(* Logix 5000 project; controller Tekno_ASRS vendor 1 type 14 code 147 rev 20.11; software revision 20.01; part 2 of 4 *)
(* tags used below, declared in another part *)
   AAxis : AXIS_CIP_DRIVE;
   AAxisMAM : MOTION_INSTRUCTION;
   AAxisMove : BOOL;
   AAxisOn : MOTION_INSTRUCTION;
   AAXisReset : MOTION_INSTRUCTION;
   AftAreaScanner : DCI_STOP;
   AftAreaZn2 : ALIAS FOR ShuttleIO:10:O.2;
   AftEndZn : BOOL;
   AftEndZnLimit : DINT;
   AftEndZone : BOOL;
   AgridLoc : DINT;
   AGVatDP : ALIAS FOR StationaryIO:1:I.3;
   AGVatPU : ALIAS FOR StationaryIO:1:I.2;
   AGVok2LvDP : ALIAS FOR StationaryIO:8:O.0;
   AGVok2LvPU : ALIAS FOR StationaryIO:8:O.1;
   AreaWarn : ALIAS FOR ShuttleIO:5:O.2;
   ASRSEnable : BOOL;
   ASRSMCR : BOOL;
   ASRSStatus : ASRS_Status;
   AutoConfig : Configuration;
   AxisStateReady : BOOL;
   BackGateInstalled : ALIAS FOR ShuttleIO:9:I.Pt01Data;
   BAxis : AXIS_CIP_DRIVE;
   BAxisMAM : MOTION_INSTRUCTION;
   BAxisMove : BOOL;
   BAXisReset : MOTION_INSTRUCTION;
   BgridLoc : DINT;
   BrakeTmr : TIMER;
   CCoordSetup : BOOL;
   CfgEnd : BayPos;
   CfgStrt : BayPos;
   CGridLoc : DINT;
   Configuration : Configuration;
   CurrentAPos : DINT;
   CurrentBPos : DINT;
   CurrentCPos : DINT;
   CurrentTask : Task;
   DemoDP : Task[3];
   DemoOns : BOOL;
   DemoPU : Task[3];
   DPCntr : DINT;
   DPReg : BOOL;
   DriveEnabled : BOOL;
   DrivesOn : BOOL;
   EStop_SafetyGate : DCI_STOP;
   FootSwitch : ALIAS FOR ShuttleIO:9:I.Pt04Data;
   ForeAreaScanner : DCI_STOP;
   ForeAreaZn2 : ALIAS FOR ShuttleIO:10:O.0;
   FrntAreaWarn : ALIAS FOR ShuttleIO:9:I.Pt00Data;
   FwdEndZn : BOOL;
   FwdEndZone : BOOL;
   GZSet : BOOL;
   GZSetEnable : BOOL;
   HighSpeedFwd : BOOL;
   HighSpeedRev : BOOL;
   HMI_Commands : HMI_Commands;
   HMIData : HMI_Data;
   HMIMsgCtrl : MESSAGE;
   HMITmr : TIMER;
   HomeSpatula : BOOL;
   Horn : ALIAS FOR ShuttleIO:5:O.1;
   JogAAxisEn : BOOL;
   JogActive : BOOL;
   JogARev : BOOL;
   JogBAxisEn : BOOL;
   JogReleaseSBrk : BOOL;
   LastAAxFlt : DINT;
   LastBAxFlt : DINT;
   LastMessageReceiveSequence : DINT;
   LiftStrainFault : BOOL;
   LiftStrainOK : BOOL;
   LoadaTask : BOOL;
   LoadTask : Task;
   LockRelease : ALIAS FOR StationaryIO:7:I.Pt04Data;
   ManConfig : Configuration;
   ManGateClosed : ALIAS FOR ShuttleIO:9:I.Pt02Data;
   ManMode : BOOL;
   ManOnBoard : ALIAS FOR ShuttleIO:5:O.5;
   MasterReset : BOOL;
   MatrixSetup : BOOL;
   MaxA : DINT;
   MaxB : DINT;
   MaxC : DINT;
   MoveComplete : BOOL;
   MoveInProcess : BOOL;
   MoveRequested : BOOL;
   MoveSafetyEnable : BOOL;
   NewAPos : DINT;
   NewBPos : DINT;
   NewCmnd : DINT;
   NewCPos : DINT;
   Override : BOOL;
   PalmButtonLeft : ALIAS FOR ShuttleIO:9:I.Pt07Data;
   PalmButtonRight : ALIAS FOR ShuttleIO:9:I.Pt06Data;
   PalmButtons : DCI_STOP;
   PorDInProc : BOOL;
   PorDStop : BOOL;
   PositionFlt : BOOL;
   PUCntr : DINT;
   Pulse : TIMER;
   PulseBit : BOOL;
   PUReg : BOOL;
   RearAreaWarn : ALIAS FOR ShuttleIO:9:I.Pt05Data;
   ReceiveMessage : Messaging;
   ReleaseSpatBrk : BOOL;
   ResetTmr : TIMER;
   RowObstruction : BOOL;
   RPE_400140 : ALIAS FOR StationaryIO:2:I.0;
   RPE_400150 : ALIAS FOR StationaryIO:2:I.1;
   RPE_400160 : ALIAS FOR StationaryIO:2:I.2;
   RPE_400170 : ALIAS FOR StationaryIO:2:I.3;
   RPE_400180 : ALIAS FOR StationaryIO:2:I.4;
   RPE_400190 : ALIAS FOR StationaryIO:2:I.5;
   RPE_400200 : ALIAS FOR StationaryIO:2:I.6;
   RPE_400210 : ALIAS FOR StationaryIO:2:I.7;
   RPE_400280 : ALIAS FOR StationaryIO:3:I.0;
   RPE_400290 : ALIAS FOR StationaryIO:3:I.1;
   RPE_400300 : ALIAS FOR StationaryIO:3:I.2;
   RPE_400310 : ALIAS FOR StationaryIO:3:I.3;
   RPE_400320 : ALIAS FOR StationaryIO:3:I.4;
   RPE_400330 : ALIAS FOR StationaryIO:3:I.5;
   RPE_400340 : ALIAS FOR StationaryIO:3:I.6;
   RPE_400350 : ALIAS FOR StationaryIO:3:I.7;
   RPE_400390 : ALIAS FOR StationaryIO:4:I.0;
   RPE_400400 : ALIAS FOR StationaryIO:4:I.1;
   RPE_400410 : ALIAS FOR StationaryIO:4:I.2;
   SafetyReset : ALIAS FOR StationaryIO:7:I.Pt03Data;
   ShuttleFault : ALIAS FOR ShuttleIO:5:O.3;
   SpatulaBrake : ALIAS FOR ShuttleIO:5:O.6;
   SpatulaHome : ALIAS FOR ShuttleIO:2:I.4;
   Start : ALIAS FOR StationaryIO:7:I.Pt02Data;
   StationaryFlt : BOOL;
   StationaryHrn : BOOL;
   StationaryMnOn : BOOL;
   StationaryRn : BOOL;
   StationaryWrn : BOOL;
   Stop : ALIAS FOR StationaryIO:7:I.Pt05Data;
   StrainFltTtl : DINT;
   SUIndPos : BOOL;
   SystemRunning : ALIAS FOR ShuttleIO:5:O.0;
   TaskFIFO : CONTROL;
   TaskFile : Task[100];
   TaskInProcess : BOOL;
   TestRun : Task[20];
   TestStop : BOOL;
   UnBindInProc : BOOL;
   XAxisBrk : ALIAS FOR ShuttleIO:5:O.4;
   XAxisEOTFlt : BOOL;
   XAxisMtrSideEOT : ALIAS FOR ShuttleIO:2:I.6;
   XAxisPnlSideEOT : ALIAS FOR ShuttleIO:2:I.7;
   XBrakeTmr : TIMER;
   XLtCTTmr : TIMER;
   XLtTTmr : TIMER;
   XPosHoldTmr : TIMER;
   XRtCTTmr : TIMER;
   XRtTTmr : TIMER;
   XStCalMode : ALIAS FOR StationaryIO:5:O.Data[0].0;
   XStrain : Strain;
   XStRunMode : ALIAS FOR StationaryIO:5:O.Data[0].1;
   XTensionOK : BOOL;
   ZAftLeftOK : BOOL;
   ZAftLtCTTmr : TIMER;
   ZAftLtTTmr : TIMER;
   ZAftRightOK : BOOL;
   ZAftRtCTTmr : TIMER;
   ZAftRtTTmr : TIMER;
   ZAftStCalMode : ALIAS FOR ShuttleIO:4:O.Data[0].0;
   ZAftStrain : Strain;
   ZAftStRunMode : ALIAS FOR ShuttleIO:4:O.Data[0].1;
   ZAxisBrk : ALIAS FOR ShuttleIO:5:O.7;
   ZAxisDnEOT : ALIAS FOR ShuttleIO:1:I.1;
   ZAxisEOTFlt : BOOL;
   ZAxisSafetyDisengage : BOOL;
   ZAxisUpEOT : ALIAS FOR ShuttleIO:1:I.0;
   ZForeLeftOK : BOOL;
   ZForeRightOK : BOOL;
   ZForeStCalMode : ALIAS FOR ShuttleIO:3:O.Data[0].0;
   ZForeStrain : Strain;
   ZForeStRunMode : ALIAS FOR ShuttleIO:3:O.Data[0].1;
   ZForLtCTTmr : TIMER;
   ZForLtTTmr : TIMER;
   ZForRtCTTmr : TIMER;
   ZForRtTTmr : TIMER;
   ZLAftLft : ALIAS FOR ShuttleIO:2:I.0;
   ZLAftRgt : ALIAS FOR ShuttleIO:2:I.1;
   ZLAutoDly : DINT;
   ZLBindTmr : TIMER;
   ZLFault : BOOL;
   ZLForeLft : ALIAS FOR ShuttleIO:2:I.3;
   ZLForeRgt : ALIAS FOR ShuttleIO:2:I.2;
   ZLManDly : DINT;
   ZLockDelay : TIMER;
   ZLsDisengaged : BOOL;
   ZLsProxOK : BOOL;
   ZPosHoldTmr : TIMER;

PROGRAM MainProgram   (* main routine MainRoutine *)
VAR
   AAxisOff : MOTION_INSTRUCTION := (FLAGS := 536870912, DN := 1, STATUS := 2, STATE := 1);
   AAxisStateMask : DINT;
   AutoMode : BOOL;
   BAxisOff : MOTION_INSTRUCTION := (FLAGS := 536870912, DN := 1, STATUS := 2, STATE := 1);
   BAxisStateMask : DINT;
   msgtest : BOOL;
   msgtest2 : BOOL;
END_VAR

ROUTINE HMI   (* ladder *)
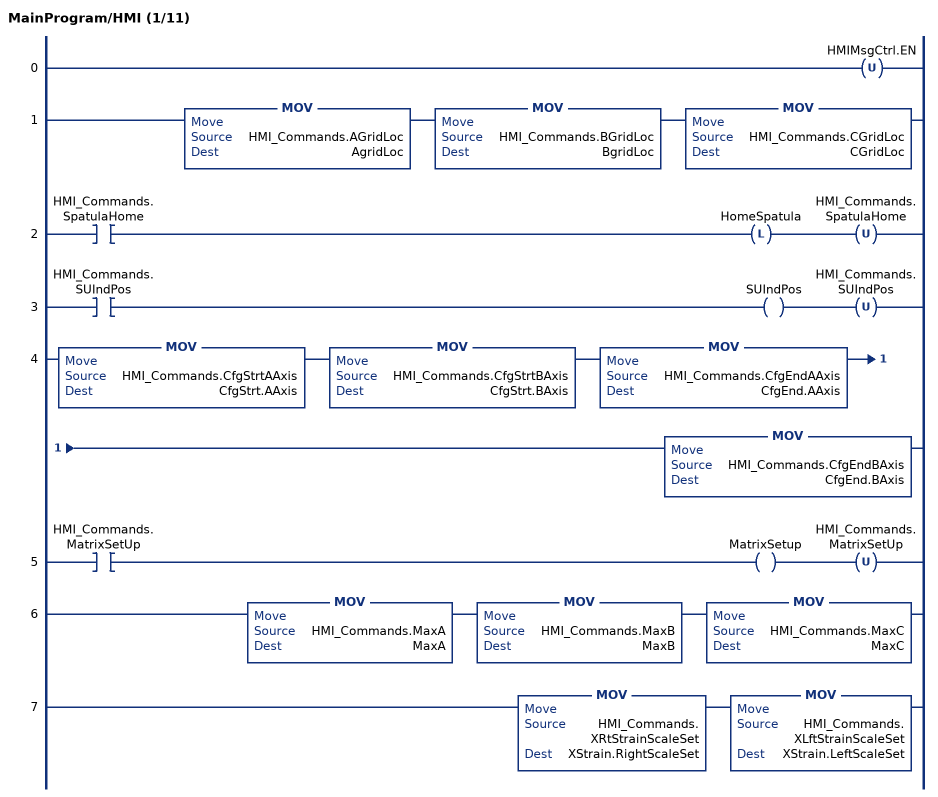
   0: OTU(HMIMsgCtrl.EN);
   1: MOV(HMI_Commands.AGridLoc,AgridLoc)MOV(HMI_Commands.BGridLoc,BgridLoc)MOV(HMI_Commands.CGridLoc,CGridLoc);
   2: XIC(HMI_Commands.SpatulaHome)OTL(HomeSpatula)OTU(HMI_Commands.SpatulaHome);
   3: XIC(HMI_Commands.SUIndPos)OTE(SUIndPos)OTU(HMI_Commands.SUIndPos);
   4: MOV(HMI_Commands.CfgStrtAAxis,CfgStrt.AAxis)MOV(HMI_Commands.CfgStrtBAxis,CfgStrt.BAxis)MOV(HMI_Commands.CfgEndAAxis,CfgEnd.AAxis)MOV(HMI_Commands.CfgEndBAxis,CfgEnd.BAxis);
   5: XIC(HMI_Commands.MatrixSetUp)OTE(MatrixSetup)OTU(HMI_Commands.MatrixSetUp);
   6: MOV(HMI_Commands.MaxA,MaxA)MOV(HMI_Commands.MaxB,MaxB)MOV(HMI_Commands.MaxC,MaxC);
   7: MOV(HMI_Commands.XRtStrainScaleSet,XStrain.RightScaleSet)MOV(HMI_Commands.XLftStrainScaleSet,XStrain.LeftScaleSet);
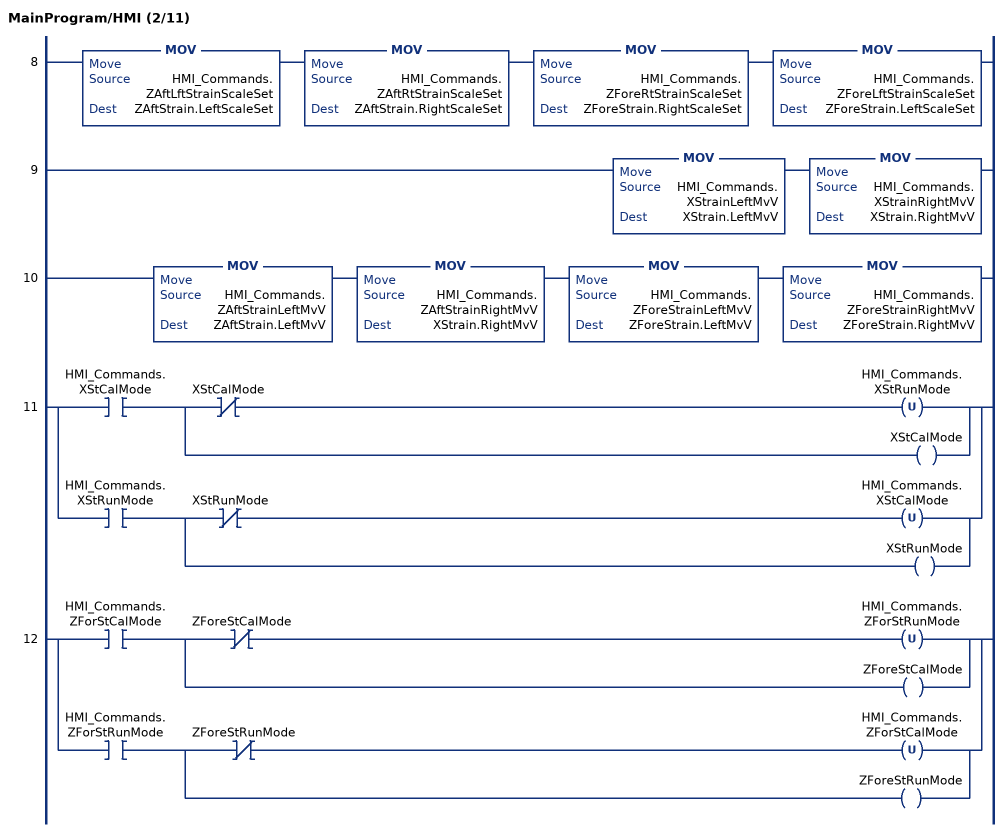
   8: MOV(HMI_Commands.ZAftLftStrainScaleSet,ZAftStrain.LeftScaleSet)MOV(HMI_Commands.ZAftRtStrainScaleSet,ZAftStrain.RightScaleSet)MOV(HMI_Commands.ZForeRtStrainScaleSet,ZForeStrain.RightScaleSet)MOV(HMI_Commands.ZForeLftStrainScaleSet,ZForeStrain.LeftScaleSet);
   9: MOV(HMI_Commands.XStrainLeftMvV,XStrain.LeftMvV)MOV(HMI_Commands.XStrainRightMvV,XStrain.RightMvV);
   10: MOV(HMI_Commands.ZAftStrainLeftMvV,ZAftStrain.LeftMvV)MOV(HMI_Commands.ZAftStrainRightMvV,XStrain.RightMvV)MOV(HMI_Commands.ZForeStrainLeftMvV,ZForeStrain.LeftMvV)MOV(HMI_Commands.ZForeStrainRightMvV,ZForeStrain.RightMvV);
   11: [XIC(HMI_Commands.XStCalMode) [XIO(XStCalMode) OTU(HMI_Commands.XStRunMode) ,OTE(XStCalMode) ] ,XIC(HMI_Commands.XStRunMode) [XIO(XStRunMode) OTU(HMI_Commands.XStCalMode) ,OTE(XStRunMode) ] ];
   12: [XIC(HMI_Commands.ZForStCalMode) [XIO(ZForeStCalMode) OTU(HMI_Commands.ZForStRunMode) ,OTE(ZForeStCalMode) ] ,XIC(HMI_Commands.ZForStRunMode) [XIO(ZForeStRunMode) OTU(HMI_Commands.ZForStCalMode) ,OTE(ZForeStRunMode) ] ];
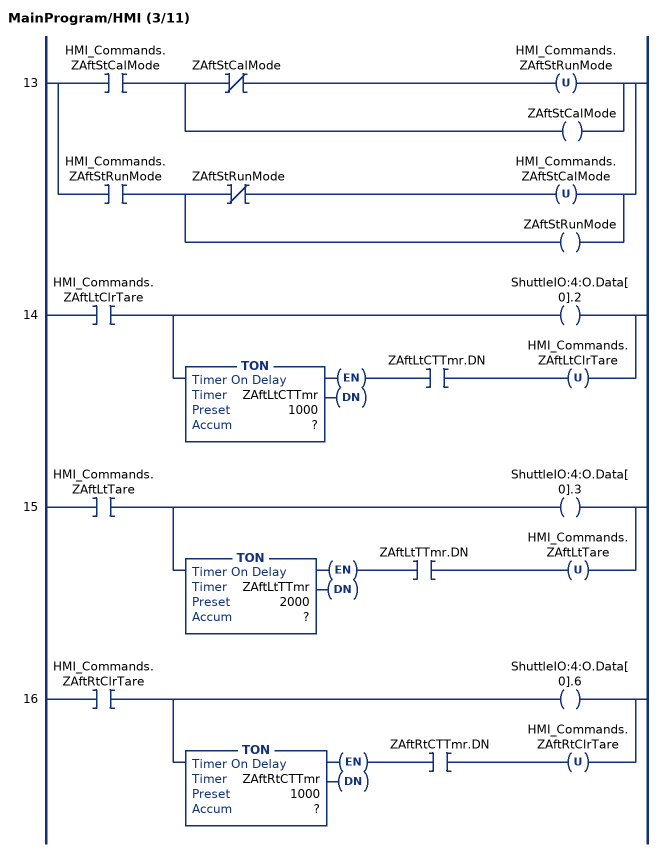
   13: [XIC(HMI_Commands.ZAftStCalMode) [XIO(ZAftStCalMode) OTU(HMI_Commands.ZAftStRunMode) ,OTE(ZAftStCalMode) ] ,XIC(HMI_Commands.ZAftStRunMode) [XIO(ZAftStRunMode) OTU(HMI_Commands.ZAftStCalMode) ,OTE(ZAftStRunMode) ] ];
   14: XIC(HMI_Commands.ZAftLtClrTare)[OTE(ShuttleIO:4:O.Data[0].2) ,TON(ZAftLtCTTmr,?,?) XIC(ZAftLtCTTmr.DN) OTU(HMI_Commands.ZAftLtClrTare) ];
   15: XIC(HMI_Commands.ZAftLtTare)[OTE(ShuttleIO:4:O.Data[0].3) ,TON(ZAftLtTTmr,?,?) XIC(ZAftLtTTmr.DN) OTU(HMI_Commands.ZAftLtTare) ];
   16: XIC(HMI_Commands.ZAftRtClrTare)[OTE(ShuttleIO:4:O.Data[0].6) ,TON(ZAftRtCTTmr,?,?) XIC(ZAftRtCTTmr.DN) OTU(HMI_Commands.ZAftRtClrTare) ];
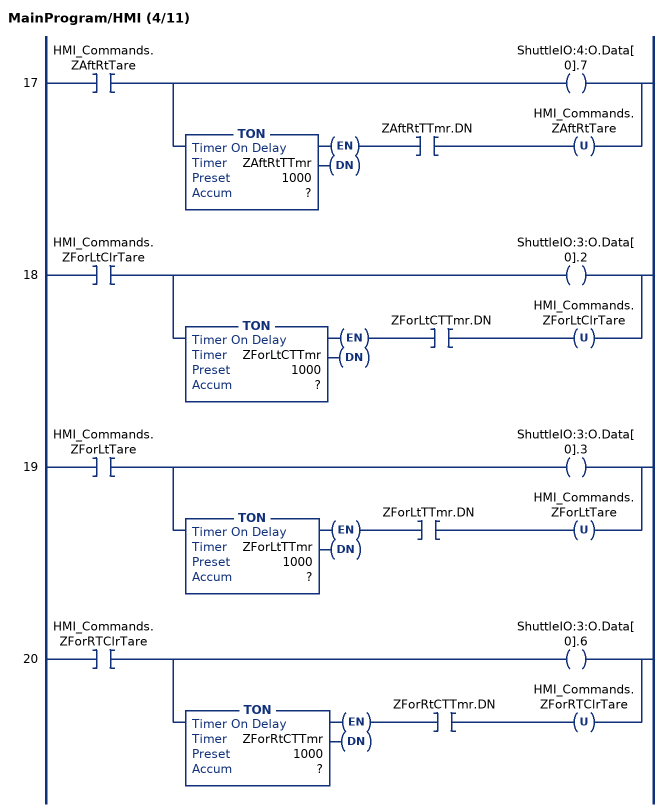
   17: XIC(HMI_Commands.ZAftRtTare)[OTE(ShuttleIO:4:O.Data[0].7) ,TON(ZAftRtTTmr,?,?) XIC(ZAftRtTTmr.DN) OTU(HMI_Commands.ZAftRtTare) ];
   18: XIC(HMI_Commands.ZForLtClrTare)[OTE(ShuttleIO:3:O.Data[0].2) ,TON(ZForLtCTTmr,?,?) XIC(ZForLtCTTmr.DN) OTU(HMI_Commands.ZForLtClrTare) ];
   19: XIC(HMI_Commands.ZForLtTare)[OTE(ShuttleIO:3:O.Data[0].3) ,TON(ZForLtTTmr,?,?) XIC(ZForLtTTmr.DN) OTU(HMI_Commands.ZForLtTare) ];
   20: XIC(HMI_Commands.ZForRTClrTare)[OTE(ShuttleIO:3:O.Data[0].6) ,TON(ZForRtCTTmr,?,?) XIC(ZForRtCTTmr.DN) OTU(HMI_Commands.ZForRTClrTare) ];
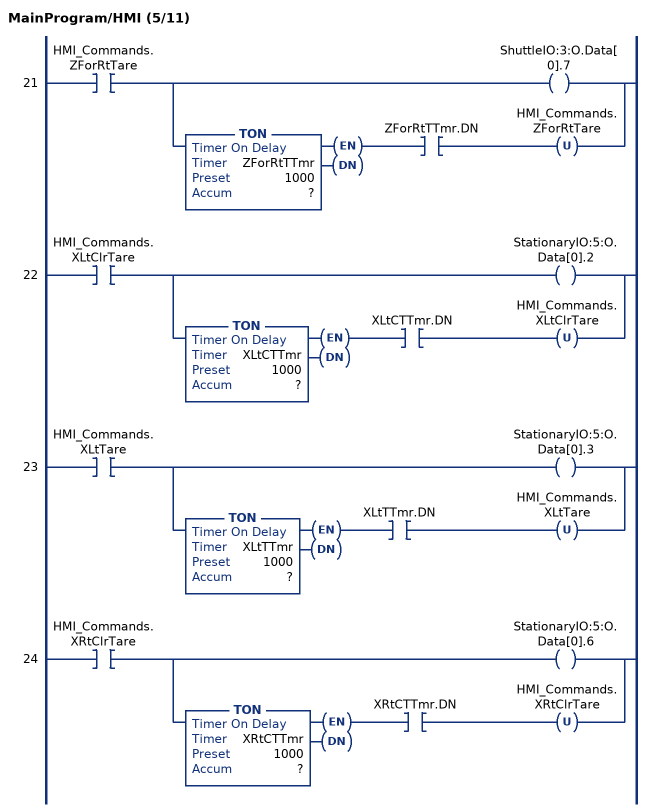
   21: XIC(HMI_Commands.ZForRtTare)[OTE(ShuttleIO:3:O.Data[0].7) ,TON(ZForRtTTmr,?,?) XIC(ZForRtTTmr.DN) OTU(HMI_Commands.ZForRtTare) ];
   22: XIC(HMI_Commands.XLtClrTare)[OTE(StationaryIO:5:O.Data[0].2) ,TON(XLtCTTmr,?,?) XIC(XLtCTTmr.DN) OTU(HMI_Commands.XLtClrTare) ];
   23: XIC(HMI_Commands.XLtTare)[OTE(StationaryIO:5:O.Data[0].3) ,TON(XLtTTmr,?,?) XIC(XLtTTmr.DN) OTU(HMI_Commands.XLtTare) ];
   24: XIC(HMI_Commands.XRtClrTare)[OTE(StationaryIO:5:O.Data[0].6) ,TON(XRtCTTmr,?,?) XIC(XRtCTTmr.DN) OTU(HMI_Commands.XRtClrTare) ];
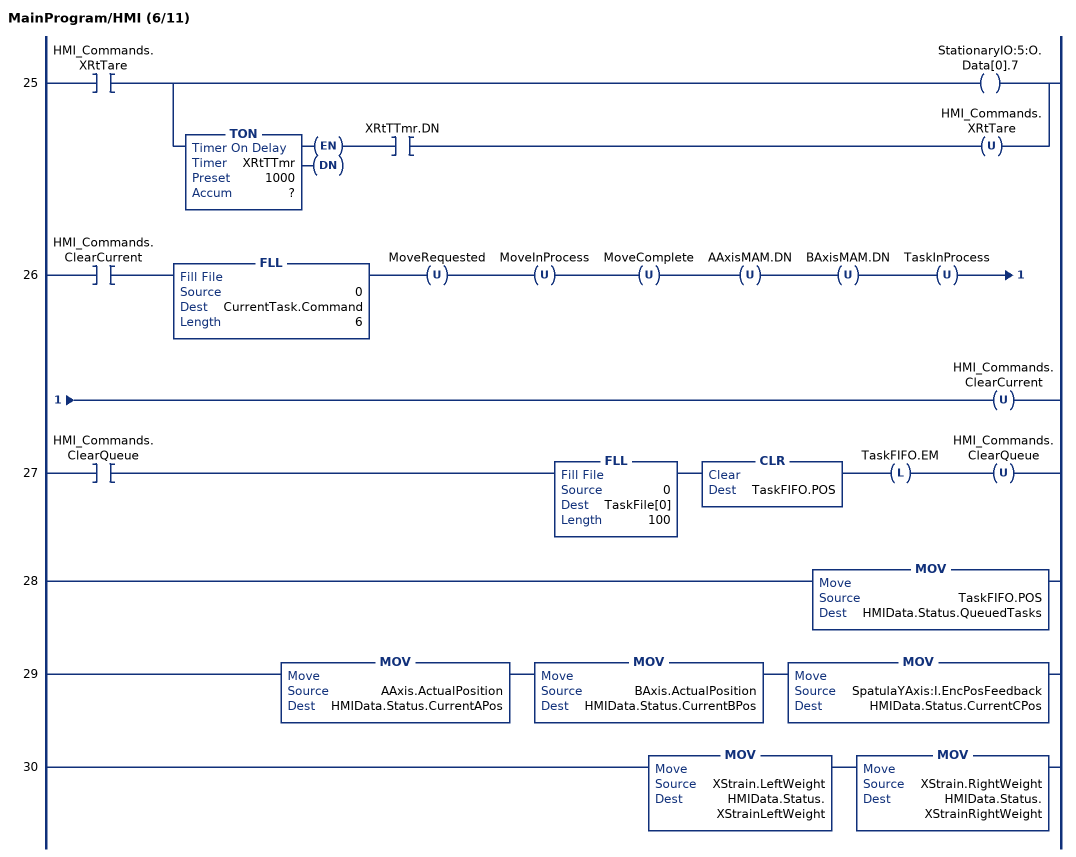
   25: XIC(HMI_Commands.XRtTare)[OTE(StationaryIO:5:O.Data[0].7) ,TON(XRtTTmr,?,?) XIC(XRtTTmr.DN) OTU(HMI_Commands.XRtTare) ];
   26: XIC(HMI_Commands.ClearCurrent)FLL(0,CurrentTask.Command,6)OTU(MoveRequested)OTU(MoveInProcess)OTU(MoveComplete)OTU(AAxisMAM.DN)OTU(BAxisMAM.DN)OTU(TaskInProcess)OTU(HMI_Commands.ClearCurrent);
   27: XIC(HMI_Commands.ClearQueue)FLL(0,TaskFile[0],100)CLR(TaskFIFO.POS)OTL(TaskFIFO.EM)OTU(HMI_Commands.ClearQueue);
   28: MOV(TaskFIFO.POS,HMIData.Status.QueuedTasks);
   29: MOV(AAxis.ActualPosition,HMIData.Status.CurrentAPos)MOV(BAxis.ActualPosition,HMIData.Status.CurrentBPos)MOV(SpatulaYAxis:I.EncPosFeedback,HMIData.Status.CurrentCPos);
   30: MOV(XStrain.LeftWeight,HMIData.Status.XStrainLeftWeight)MOV(XStrain.RightWeight,HMIData.Status.XStrainRightWeight);
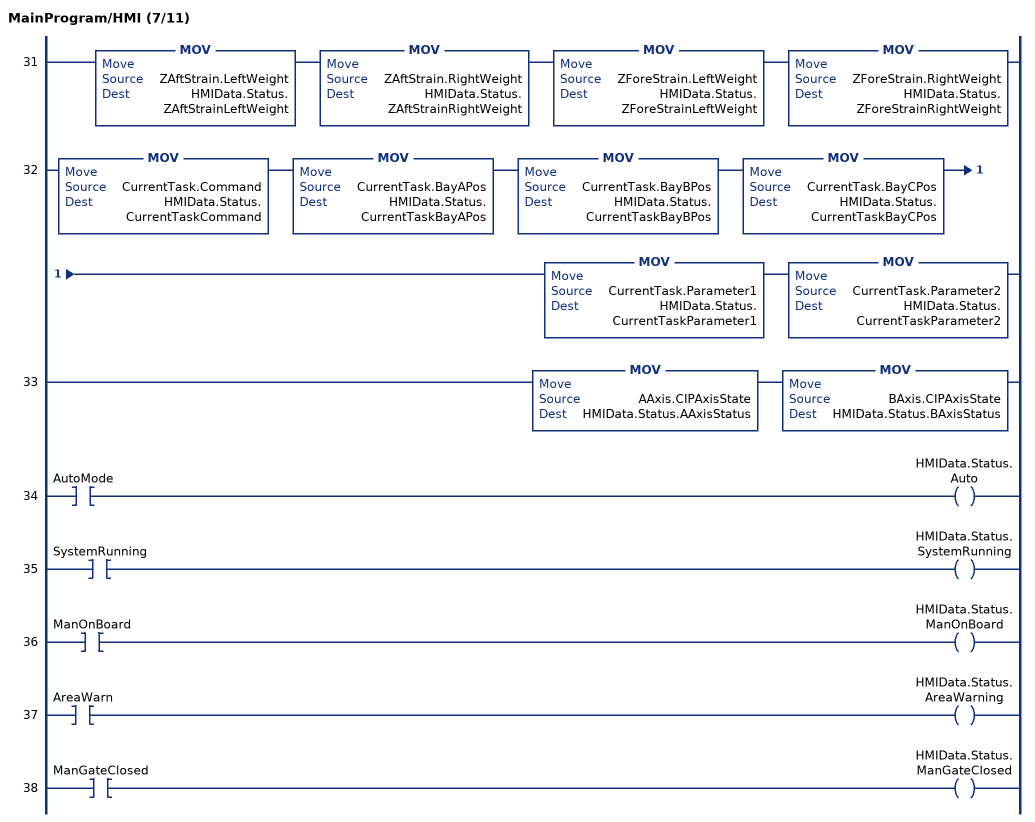
   31: MOV(ZAftStrain.LeftWeight,HMIData.Status.ZAftStrainLeftWeight)MOV(ZAftStrain.RightWeight,HMIData.Status.ZAftStrainRightWeight)MOV(ZForeStrain.LeftWeight,HMIData.Status.ZForeStrainLeftWeight)MOV(ZForeStrain.RightWeight,HMIData.Status.ZForeStrainRightWeight);
   32: MOV(CurrentTask.Command,HMIData.Status.CurrentTaskCommand)MOV(CurrentTask.BayAPos,HMIData.Status.CurrentTaskBayAPos)MOV(CurrentTask.BayBPos,HMIData.Status.CurrentTaskBayBPos)MOV(CurrentTask.BayCPos,HMIData.Status.CurrentTaskBayCPos)MOV(CurrentTask.Parameter1,HMIData.Status.CurrentTaskParameter1)MOV(CurrentTask.Parameter2,HMIData.Status.CurrentTaskParameter2);
   33: MOV(AAxis.CIPAxisState,HMIData.Status.AAxisStatus)MOV(BAxis.CIPAxisState,HMIData.Status.BAxisStatus);
   34: XIC(AutoMode)OTE(HMIData.Status.Auto);
   35: XIC(SystemRunning)OTE(HMIData.Status.SystemRunning);
   36: XIC(ManOnBoard)OTE(HMIData.Status.ManOnBoard);
   37: XIC(AreaWarn)OTE(HMIData.Status.AreaWarning);
   38: XIC(ManGateClosed)OTE(HMIData.Status.ManGateClosed);
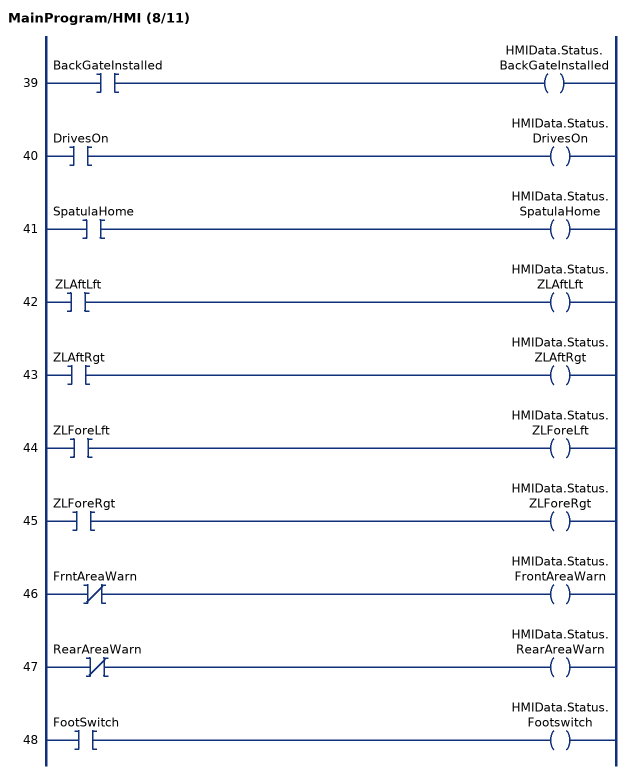
   39: XIC(BackGateInstalled)OTE(HMIData.Status.BackGateInstalled);
   40: XIC(DrivesOn)OTE(HMIData.Status.DrivesOn);
   41: XIC(SpatulaHome)OTE(HMIData.Status.SpatulaHome);
   42: XIC(ZLAftLft)OTE(HMIData.Status.ZLAftLft);
   43: XIC(ZLAftRgt)OTE(HMIData.Status.ZLAftRgt);
   44: XIC(ZLForeLft)OTE(HMIData.Status.ZLForeLft);
   45: XIC(ZLForeRgt)OTE(HMIData.Status.ZLForeRgt);
   46: XIO(FrntAreaWarn)OTE(HMIData.Status.FrontAreaWarn);
   47: XIO(RearAreaWarn)OTE(HMIData.Status.RearAreaWarn);
   48: XIC(FootSwitch)OTE(HMIData.Status.Footswitch);
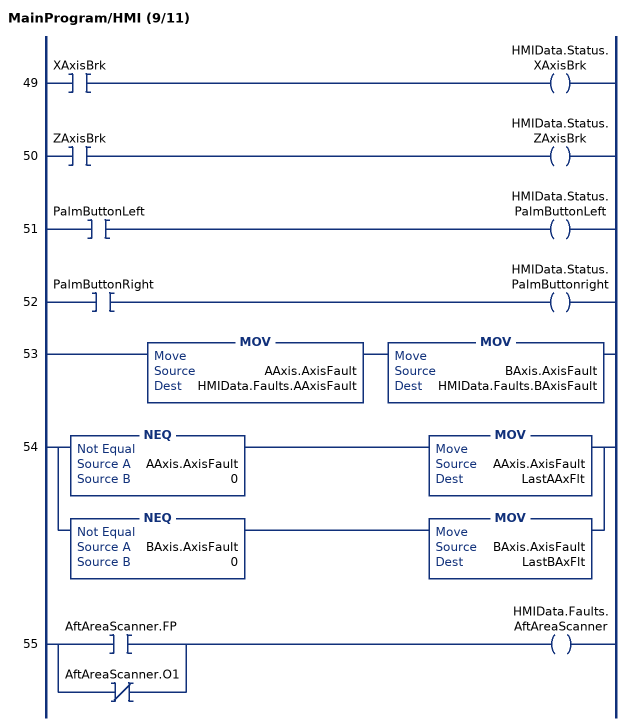
   49: XIC(XAxisBrk)OTE(HMIData.Status.XAxisBrk);
   50: XIC(ZAxisBrk)OTE(HMIData.Status.ZAxisBrk);
   51: XIC(PalmButtonLeft)OTE(HMIData.Status.PalmButtonLeft);
   52: XIC(PalmButtonRight)OTE(HMIData.Status.PalmButtonright);
   53: MOV(AAxis.AxisFault,HMIData.Faults.AAxisFault)MOV(BAxis.AxisFault,HMIData.Faults.BAxisFault);
   54: [NEQ(AAxis.AxisFault,0) MOV(AAxis.AxisFault,LastAAxFlt) ,NEQ(BAxis.AxisFault,0) MOV(BAxis.AxisFault,LastBAxFlt) ];
   55: [XIC(AftAreaScanner.FP) ,XIO(AftAreaScanner.O1) ]OTE(HMIData.Faults.AftAreaScanner);
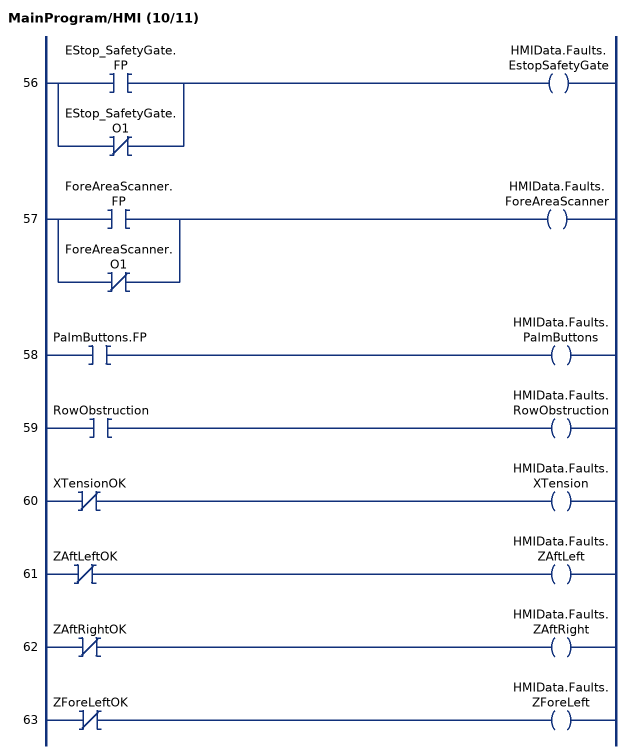
   56: [XIC(EStop_SafetyGate.FP) ,XIO(EStop_SafetyGate.O1) ]OTE(HMIData.Faults.EstopSafetyGate);
   57: [XIC(ForeAreaScanner.FP) ,XIO(ForeAreaScanner.O1) ]OTE(HMIData.Faults.ForeAreaScanner);
   58: XIC(PalmButtons.FP)OTE(HMIData.Faults.PalmButtons);
   59: XIC(RowObstruction)OTE(HMIData.Faults.RowObstruction);
   60: XIO(XTensionOK)OTE(HMIData.Faults.XTension);
   61: XIO(ZAftLeftOK)OTE(HMIData.Faults.ZAftLeft);
   62: XIO(ZAftRightOK)OTE(HMIData.Faults.ZAftRight);
   63: XIO(ZForeLeftOK)OTE(HMIData.Faults.ZForeLeft);
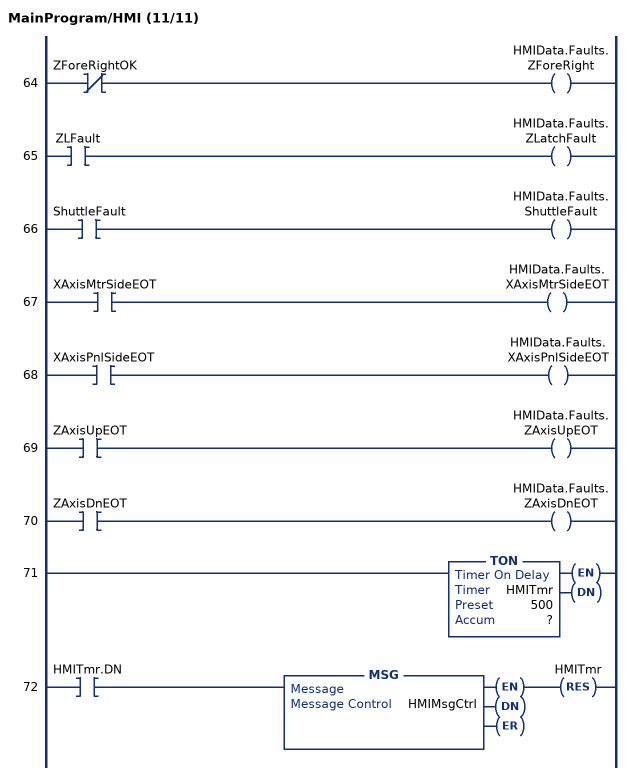
   64: XIO(ZForeRightOK)OTE(HMIData.Faults.ZForeRight);
   65: XIC(ZLFault)OTE(HMIData.Faults.ZLatchFault);
   66: XIC(ShuttleFault)OTE(HMIData.Faults.ShuttleFault);
   67: XIC(XAxisMtrSideEOT)OTE(HMIData.Faults.XAxisMtrSideEOT);
   68: XIC(XAxisPnlSideEOT)OTE(HMIData.Faults.XAxisPnlSideEOT);
   69: XIC(ZAxisUpEOT)OTE(HMIData.Faults.ZAxisUpEOT);
   70: XIC(ZAxisDnEOT)OTE(HMIData.Faults.ZAxisDnEOT);
   71: TON(HMITmr,?,?);
   72: XIC(HMITmr.DN)MSG(HMIMsgCtrl)RES(HMITmr);
END_ROUTINE

ROUTINE MainRoutine   (* ladder *)
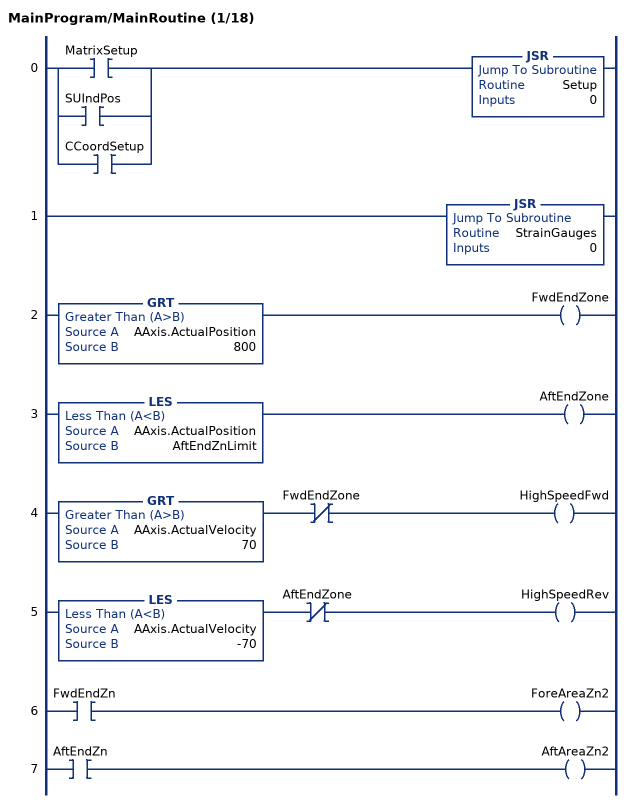
   0: [XIC(MatrixSetup) ,XIC(SUIndPos) ,XIC(CCoordSetup) ]JSR(Setup,0);
   1: JSR(StrainGauges,0);
   2: GRT(AAxis.ActualPosition,800)OTE(FwdEndZone);
   3: LES(AAxis.ActualPosition,AftEndZnLimit)OTE(AftEndZone);
   4: GRT(AAxis.ActualVelocity,70)XIO(FwdEndZone)OTE(HighSpeedFwd);
   5: LES(AAxis.ActualVelocity,-70)XIO(AftEndZone)OTE(HighSpeedRev);
   6: XIC(FwdEndZn)OTE(ForeAreaZn2);
   7: XIC(AftEndZn)OTE(AftAreaZn2);
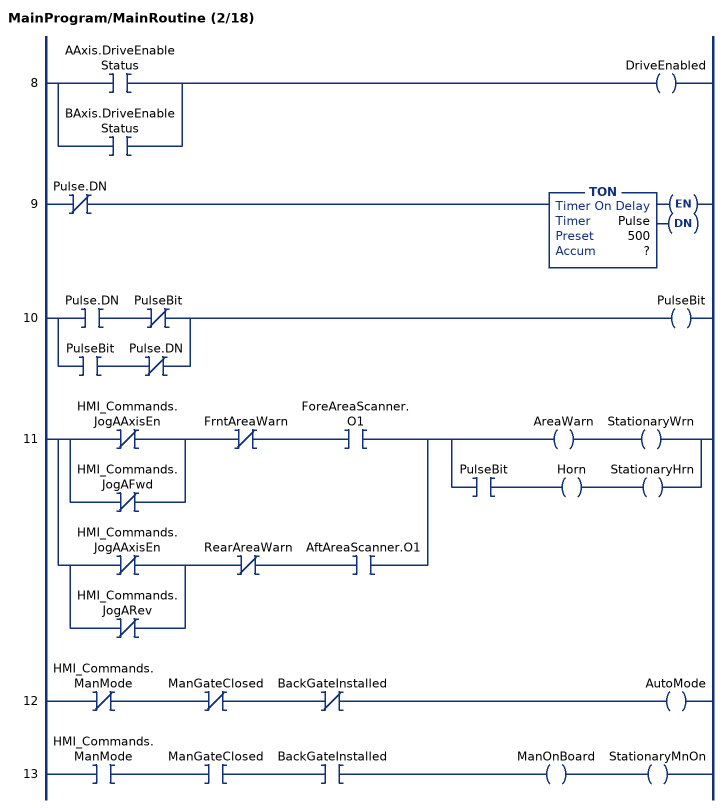
   8: [XIC(AAxis.DriveEnableStatus) ,XIC(BAxis.DriveEnableStatus) ]OTE(DriveEnabled);
   9: XIO(Pulse.DN)TON(Pulse,?,?);
   10: [XIC(Pulse.DN) XIO(PulseBit) ,XIC(PulseBit) XIO(Pulse.DN) ]OTE(PulseBit);
   11: [[XIO(HMI_Commands.JogAAxisEn) ,XIO(HMI_Commands.JogAFwd) ] XIO(FrntAreaWarn) XIC(ForeAreaScanner.O1) ,[XIO(HMI_Commands.JogAAxisEn) ,XIO(HMI_Commands.JogARev) ] XIO(RearAreaWarn) XIC(AftAreaScanner.O1) ][OTE(AreaWarn) OTE(StationaryWrn) ,XIC(PulseBit) OTE(Horn) OTE(StationaryHrn) ];
   12: XIO(HMI_Commands.ManMode)XIO(ManGateClosed)XIO(BackGateInstalled)OTE(AutoMode);
   13: XIC(HMI_Commands.ManMode)XIC(ManGateClosed)XIC(BackGateInstalled)OTE(ManOnBoard)OTE(StationaryMnOn);
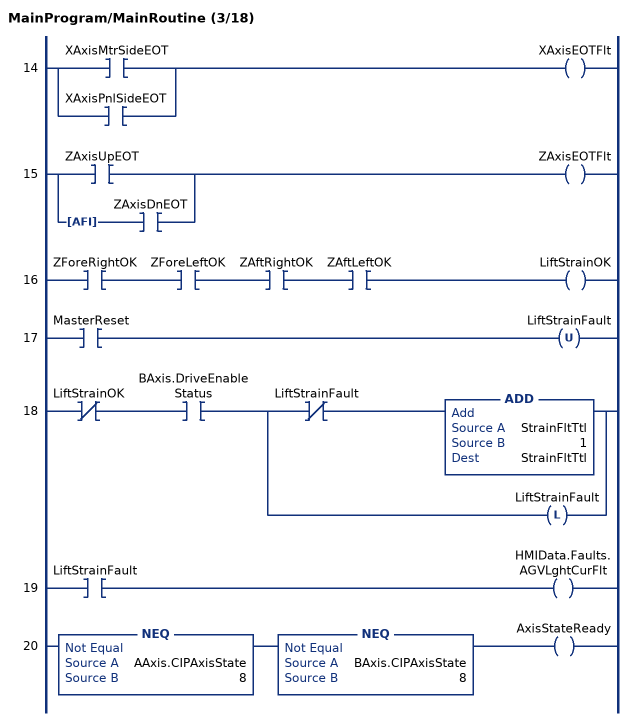
   14: [XIC(XAxisMtrSideEOT) ,XIC(XAxisPnlSideEOT) ]OTE(XAxisEOTFlt);
   15: [XIC(ZAxisUpEOT) ,AFI() XIC(ZAxisDnEOT) ]OTE(ZAxisEOTFlt);
   16: XIC(ZForeRightOK)XIC(ZForeLeftOK)XIC(ZAftRightOK)XIC(ZAftLeftOK)OTE(LiftStrainOK);
   17: XIC(MasterReset)OTU(LiftStrainFault);
   18: XIO(LiftStrainOK)XIC(BAxis.DriveEnableStatus)[XIO(LiftStrainFault) ADD(StrainFltTtl,1,StrainFltTtl) ,OTL(LiftStrainFault) ];
   19: XIC(LiftStrainFault)OTE(HMIData.Faults.AGVLghtCurFlt);
   20: NEQ(AAxis.CIPAxisState,8)NEQ(BAxis.CIPAxisState,8)OTE(AxisStateReady);
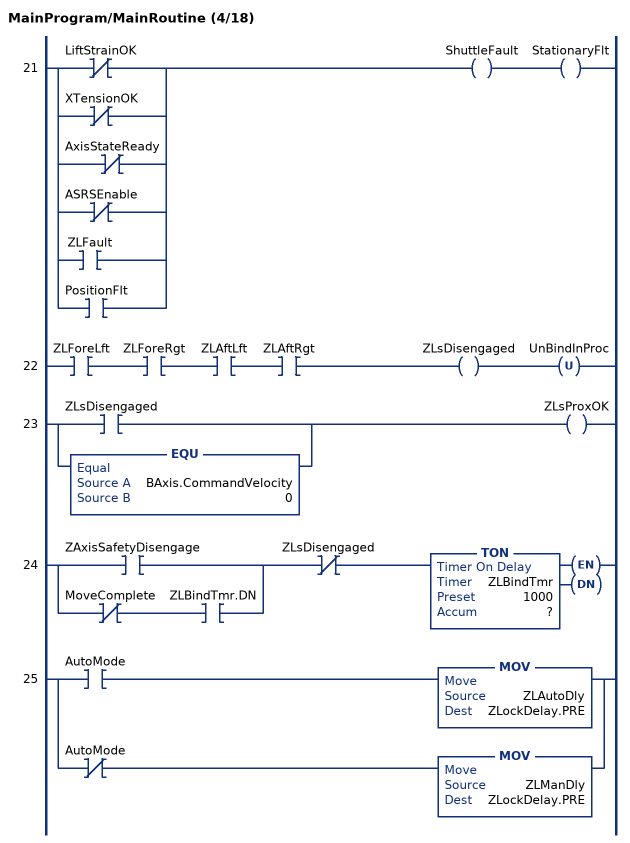
   21: [XIO(LiftStrainOK) ,XIO(XTensionOK) ,XIO(AxisStateReady) ,XIO(ASRSEnable) ,XIC(ZLFault) ,XIC(PositionFlt) ]OTE(ShuttleFault)OTE(StationaryFlt);
   22: XIC(ZLForeLft)XIC(ZLForeRgt)XIC(ZLAftLft)XIC(ZLAftRgt)OTE(ZLsDisengaged)OTU(UnBindInProc);
   23: [XIC(ZLsDisengaged) ,EQU(BAxis.CommandVelocity,0) ]OTE(ZLsProxOK);
   24: [XIC(ZAxisSafetyDisengage) ,XIO(MoveComplete) XIC(ZLBindTmr.DN) ]XIO(ZLsDisengaged)TON(ZLBindTmr,?,?);
   25: [XIC(AutoMode) MOV(ZLAutoDly,ZLockDelay.PRE) ,XIO(AutoMode) MOV(ZLManDly,ZLockDelay.PRE) ];
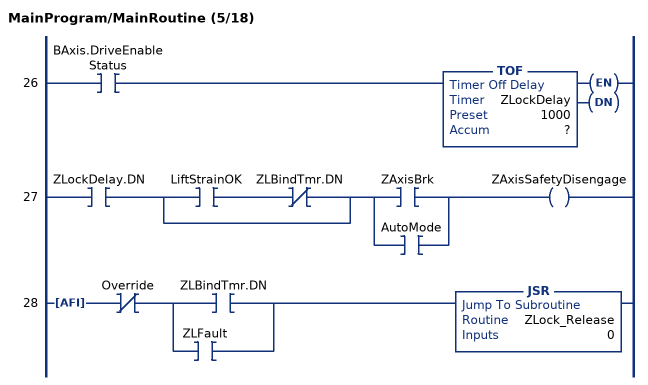
   26: XIC(BAxis.DriveEnableStatus)TOF(ZLockDelay,?,?);
   27: XIC(ZLockDelay.DN)[XIC(LiftStrainOK) XIO(ZLBindTmr.DN) ,][XIC(ZAxisBrk) ,XIC(AutoMode) ]OTE(ZAxisSafetyDisengage);
   28: AFI()XIO(Override)[XIC(ZLBindTmr.DN) ,XIC(ZLFault) ]JSR(ZLock_Release,0);
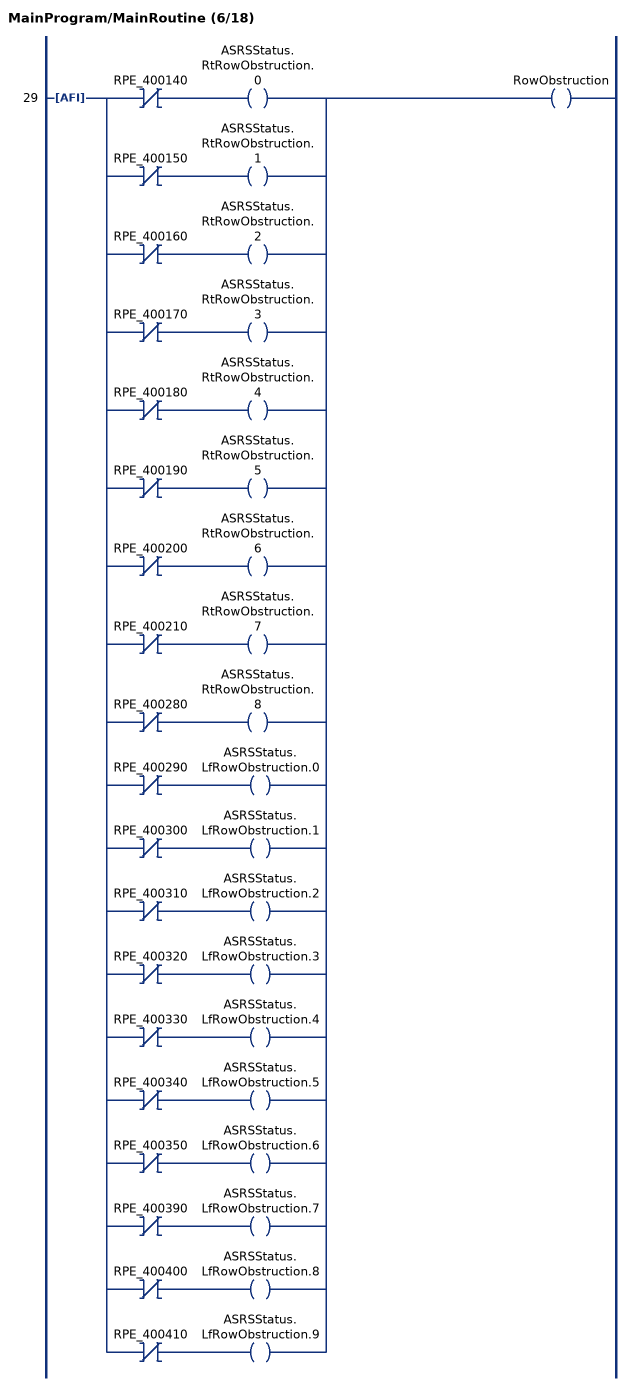
   29: AFI()[XIO(RPE_400140) OTE(ASRSStatus.RtRowObstruction.0) ,XIO(RPE_400150) OTE(ASRSStatus.RtRowObstruction.1) ,XIO(RPE_400160) OTE(ASRSStatus.RtRowObstruction.2) ,XIO(RPE_400170) OTE(ASRSStatus.RtRowObstruction.3) ,XIO(RPE_400180) OTE(ASRSStatus.RtRowObstruction.4) ,XIO(RPE_400190) OTE(ASRSStatus.RtRowObstruction.5) ,XIO(RPE_400200) OTE(ASRSStatus.RtRowObstruction.6) ,XIO(RPE_400210) OTE(ASRSStatus.RtRowObstruction.7) ,XIO(RPE_400280) OTE(ASRSStatus.RtRowObstruction.8) ,XIO(RPE_400290) OTE(ASRSStatus.LfRowObstruction.0) ,XIO(RPE_400300) OTE(ASRSStatus.LfRowObstruction.1) ,XIO(RPE_400310) OTE(ASRSStatus.LfRowObstruction.2) ,XIO(RPE_400320) OTE(ASRSStatus.LfRowObstruction.3) ,XIO(RPE_400330) OTE(ASRSStatus.LfRowObstruction.4) ,XIO(RPE_400340) OTE(ASRSStatus.LfRowObstruction.5) ,XIO(RPE_400350) OTE(ASRSStatus.LfRowObstruction.6) ,XIO(RPE_400390) OTE(ASRSStatus.LfRowObstruction.7) ,XIO(RPE_400400) OTE(ASRSStatus.LfRowObstruction.8) ,XIO(RPE_400410) OTE(ASRSStatus.LfRowObstruction.9) ]OTE(RowObstruction);
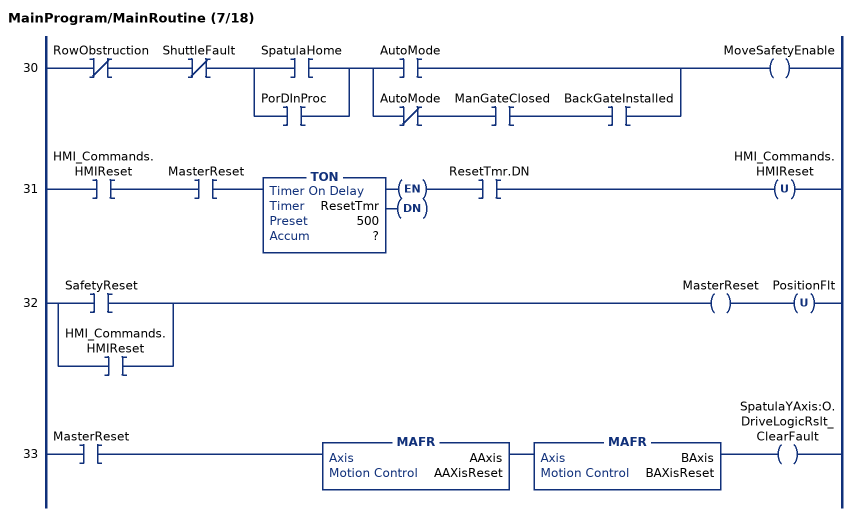
   30: XIO(RowObstruction)XIO(ShuttleFault)[XIC(SpatulaHome) ,XIC(PorDInProc) ][XIC(AutoMode) ,XIO(AutoMode) XIC(ManGateClosed) XIC(BackGateInstalled) ]OTE(MoveSafetyEnable);
   31: XIC(HMI_Commands.HMIReset)XIC(MasterReset)TON(ResetTmr,?,?)XIC(ResetTmr.DN)OTU(HMI_Commands.HMIReset);
   32: [XIC(SafetyReset) ,XIC(HMI_Commands.HMIReset) ]OTE(MasterReset)OTU(PositionFlt);
   33: XIC(MasterReset)MAFR(AAxis,AAXisReset)MAFR(BAxis,BAXisReset)OTE(SpatulaYAxis:O.DriveLogicRslt_ClearFault);
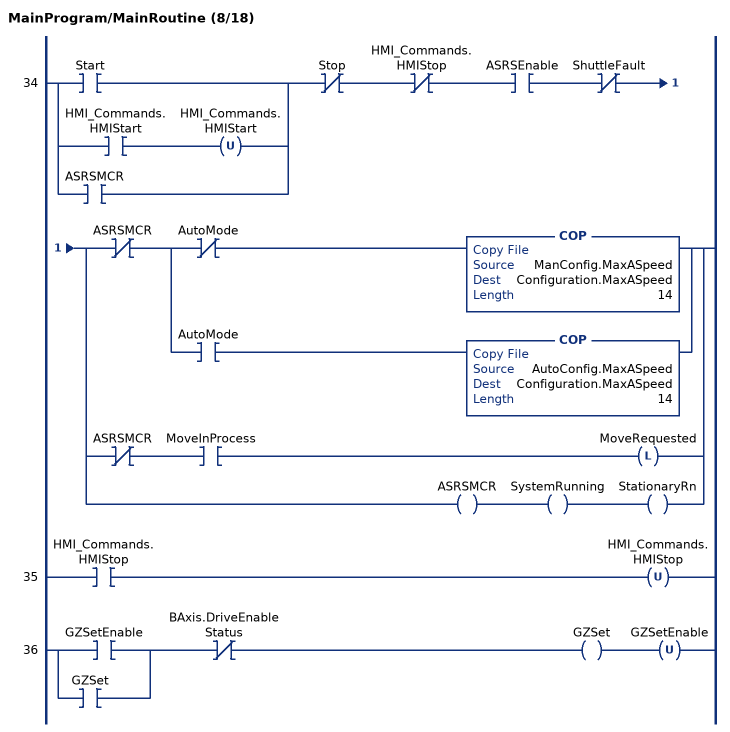
   34: [XIC(Start) ,XIC(HMI_Commands.HMIStart) OTU(HMI_Commands.HMIStart) ,XIC(ASRSMCR) ]XIO(Stop)XIO(HMI_Commands.HMIStop)XIC(ASRSEnable)XIO(ShuttleFault)[XIO(ASRSMCR) [XIO(AutoMode) COP(ManConfig.MaxASpeed,Configuration.MaxASpeed,14) ,XIC(AutoMode) COP(AutoConfig.MaxASpeed,Configuration.MaxASpeed,14) ] ,XIO(ASRSMCR) XIC(MoveInProcess) OTL(MoveRequested) ,OTE(ASRSMCR) OTE(SystemRunning) OTE(StationaryRn) ];
   35: XIC(HMI_Commands.HMIStop)OTU(HMI_Commands.HMIStop);
   36: [XIC(GZSetEnable) ,XIC(GZSet) ]XIO(BAxis.DriveEnableStatus)OTE(GZSet)OTU(GZSetEnable);
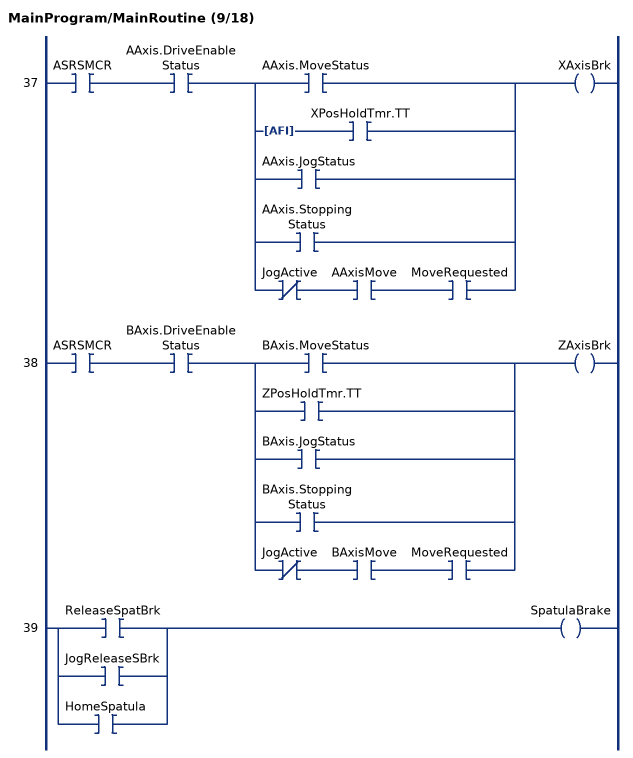
   37: XIC(ASRSMCR)XIC(AAxis.DriveEnableStatus)[XIC(AAxis.MoveStatus) ,AFI() XIC(XPosHoldTmr.TT) ,XIC(AAxis.JogStatus) ,XIC(AAxis.StoppingStatus) ,XIO(JogActive) XIC(AAxisMove) XIC(MoveRequested) ]OTE(XAxisBrk);
   38: XIC(ASRSMCR)XIC(BAxis.DriveEnableStatus)[XIC(BAxis.MoveStatus) ,XIC(ZPosHoldTmr.TT) ,XIC(BAxis.JogStatus) ,XIC(BAxis.StoppingStatus) ,XIO(JogActive) XIC(BAxisMove) XIC(MoveRequested) ]OTE(ZAxisBrk);
   39: [XIC(ReleaseSpatBrk) ,XIC(JogReleaseSBrk) ,XIC(HomeSpatula) ]OTE(SpatulaBrake);
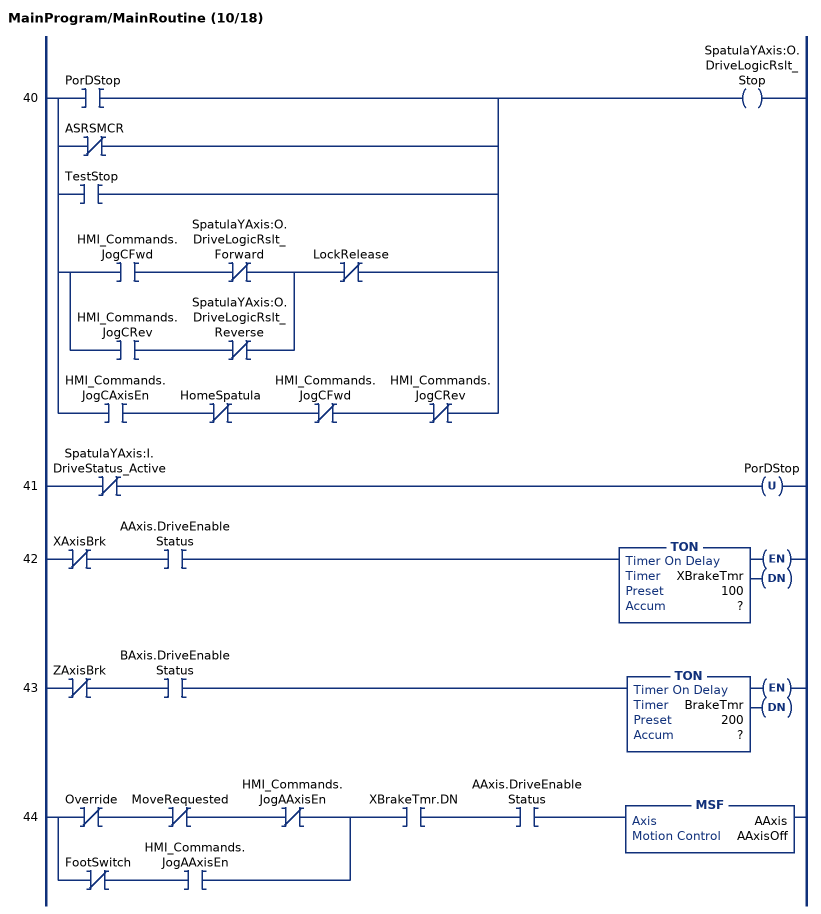
   40: [XIC(PorDStop) ,XIO(ASRSMCR) ,XIC(TestStop) ,[XIC(HMI_Commands.JogCFwd) XIO(SpatulaYAxis:O.DriveLogicRslt_Forward) ,XIC(HMI_Commands.JogCRev) XIO(SpatulaYAxis:O.DriveLogicRslt_Reverse) ] XIO(LockRelease) ,XIC(HMI_Commands.JogCAxisEn) XIO(HomeSpatula) XIO(HMI_Commands.JogCFwd) XIO(HMI_Commands.JogCRev) ]OTE(SpatulaYAxis:O.DriveLogicRslt_Stop);
   41: XIO(SpatulaYAxis:I.DriveStatus_Active)OTU(PorDStop);
   42: XIO(XAxisBrk)XIC(AAxis.DriveEnableStatus)TON(XBrakeTmr,?,?);
   43: XIO(ZAxisBrk)XIC(BAxis.DriveEnableStatus)TON(BrakeTmr,?,?);
   44: [XIO(Override) XIO(MoveRequested) XIO(HMI_Commands.JogAAxisEn) ,XIO(FootSwitch) XIC(HMI_Commands.JogAAxisEn) ]XIC(XBrakeTmr.DN)XIC(AAxis.DriveEnableStatus)MSF(AAxis,AAxisOff);
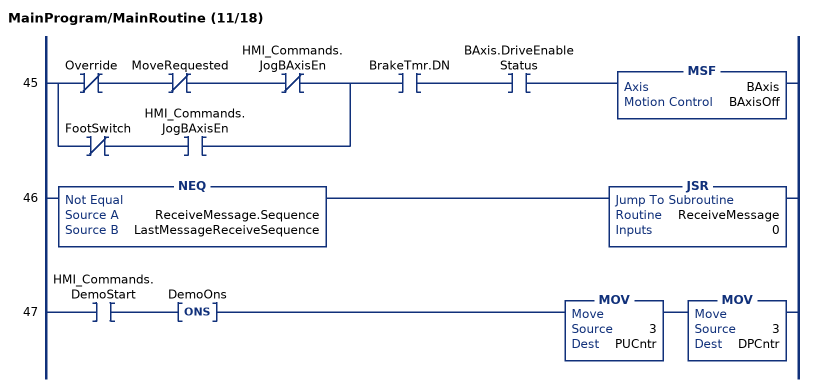
   45: [XIO(Override) XIO(MoveRequested) XIO(HMI_Commands.JogBAxisEn) ,XIO(FootSwitch) XIC(HMI_Commands.JogBAxisEn) ]XIC(BrakeTmr.DN)XIC(BAxis.DriveEnableStatus)MSF(BAxis,BAxisOff);
   46: NEQ(ReceiveMessage.Sequence,LastMessageReceiveSequence)JSR(ReceiveMessage,0);
   47: XIC(HMI_Commands.DemoStart)ONS(DemoOns)MOV(3,PUCntr)MOV(3,DPCntr);
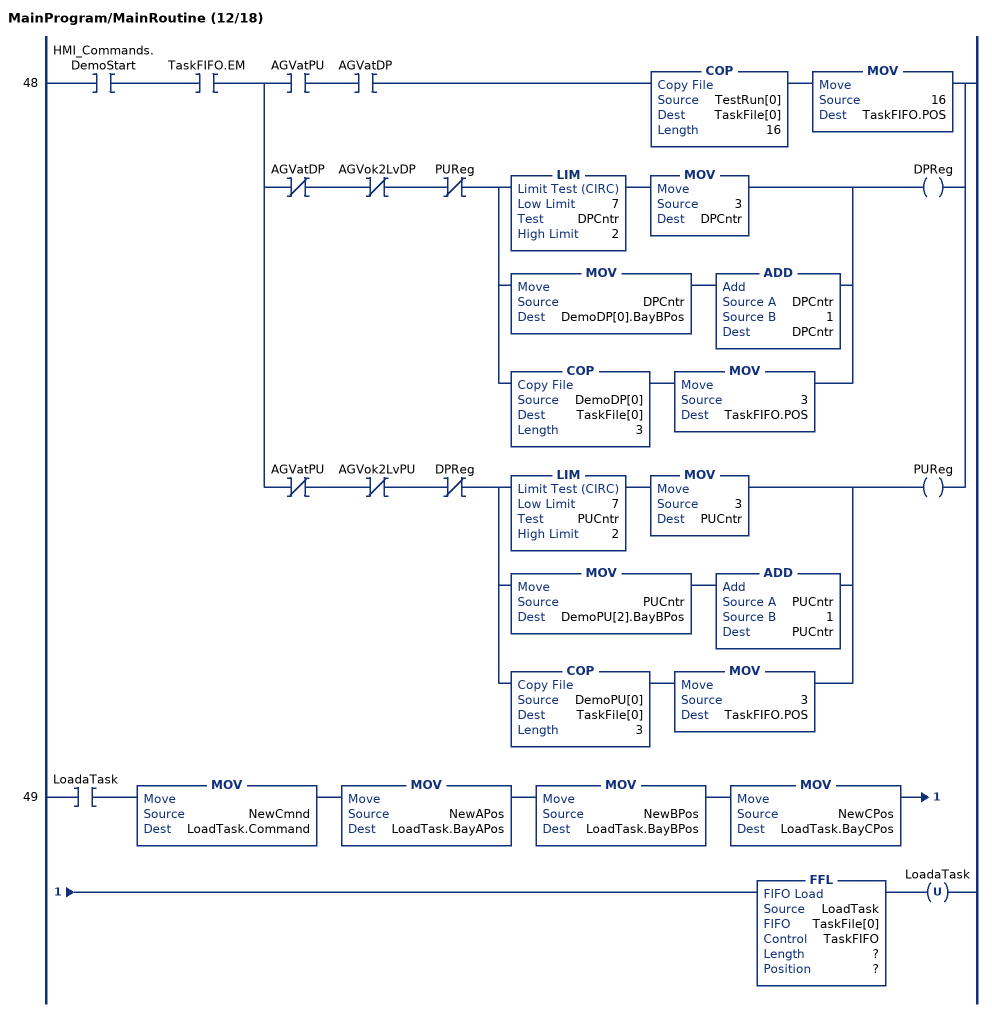
   48: XIC(HMI_Commands.DemoStart)XIC(TaskFIFO.EM)[XIC(AGVatPU) XIC(AGVatDP) COP(TestRun[0],TaskFile[0],16) MOV(16,TaskFIFO.POS) ,XIO(AGVatDP) XIO(AGVok2LvDP) XIO(PUReg) [LIM(7,DPCntr,2) MOV(3,DPCntr) ,MOV(DPCntr,DemoDP[0].BayBPos) ADD(DPCntr,1,DPCntr) ,COP(DemoDP[0],TaskFile[0],3) MOV(3,TaskFIFO.POS) ] OTE(DPReg) ,XIO(AGVatPU) XIO(AGVok2LvPU) XIO(DPReg) [LIM(7,PUCntr,2) MOV(3,PUCntr) ,MOV(PUCntr,DemoPU[2].BayBPos) ADD(PUCntr,1,PUCntr) ,COP(DemoPU[0],TaskFile[0],3) MOV(3,TaskFIFO.POS) ] OTE(PUReg) ];
   49: XIC(LoadaTask)MOV(NewCmnd,LoadTask.Command)MOV(NewAPos,LoadTask.BayAPos)MOV(NewBPos,LoadTask.BayBPos)MOV(NewCPos,LoadTask.BayCPos)FFL(LoadTask,TaskFile[0],TaskFIFO,?,?)OTU(LoadaTask);
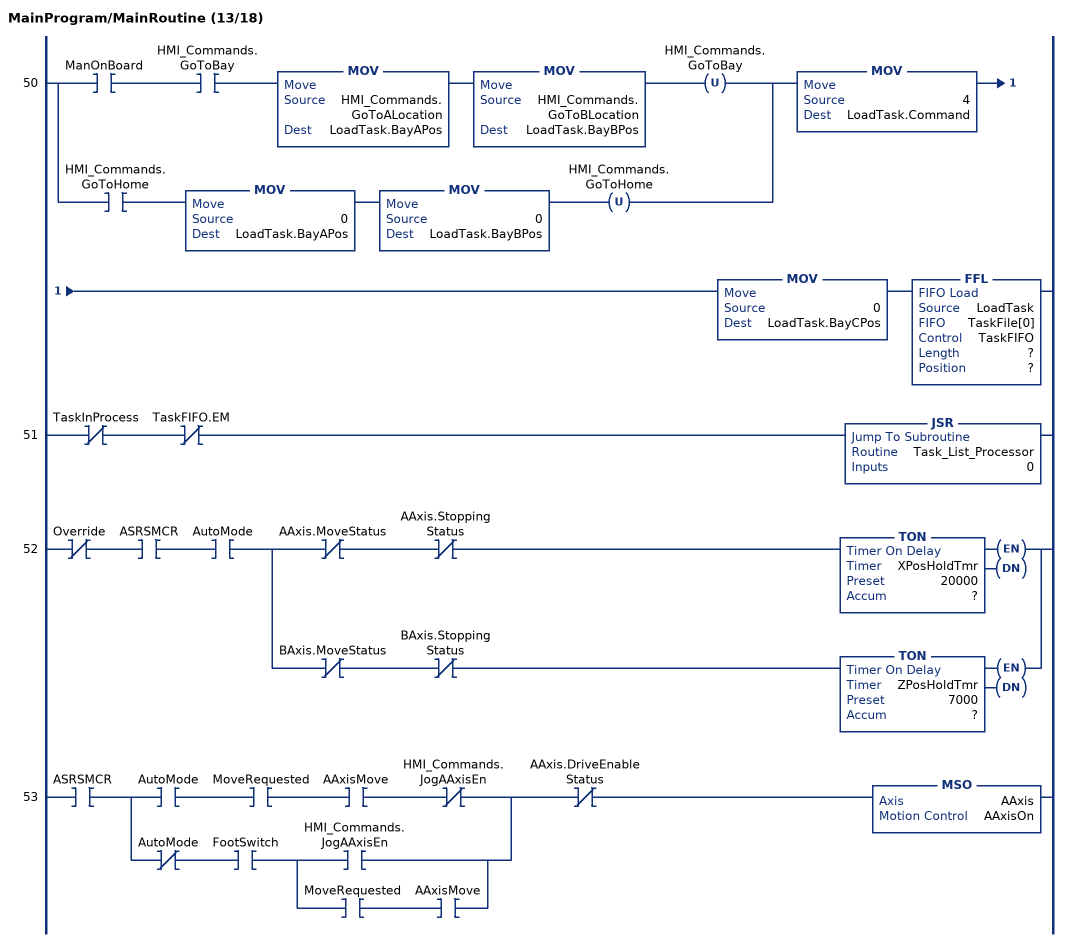
   50: [XIC(ManOnBoard) XIC(HMI_Commands.GoToBay) MOV(HMI_Commands.GoToALocation,LoadTask.BayAPos) MOV(HMI_Commands.GoToBLocation,LoadTask.BayBPos) OTU(HMI_Commands.GoToBay) ,XIC(HMI_Commands.GoToHome) MOV(0,LoadTask.BayAPos) MOV(0,LoadTask.BayBPos) OTU(HMI_Commands.GoToHome) ]MOV(4,LoadTask.Command)MOV(0,LoadTask.BayCPos)FFL(LoadTask,TaskFile[0],TaskFIFO,?,?);
   51: XIO(TaskInProcess)XIO(TaskFIFO.EM)JSR(Task_List_Processor,0);
   52: XIO(Override)XIC(ASRSMCR)XIC(AutoMode)[XIO(AAxis.MoveStatus) XIO(AAxis.StoppingStatus) TON(XPosHoldTmr,?,?) ,XIO(BAxis.MoveStatus) XIO(BAxis.StoppingStatus) TON(ZPosHoldTmr,?,?) ];
   53: XIC(ASRSMCR)[XIC(AutoMode) XIC(MoveRequested) XIC(AAxisMove) XIO(HMI_Commands.JogAAxisEn) ,XIO(AutoMode) XIC(FootSwitch) [XIC(HMI_Commands.JogAAxisEn) ,XIC(MoveRequested) XIC(AAxisMove) ] ]XIO(AAxis.DriveEnableStatus)MSO(AAxis,AAxisOn);
